TYPE Response_Values :
STRUCT
	Header				:UINT;			// Fixed 0x1234
	Status				:UINT;			// Status word of the sensor and Compute Box
	Fx					:INT;			// X-axis force in 32 bit Counts*
	Fy					:INT;			// Y-axis force in 32 bit Counts*
	Fz					:INT;			// Z-axis force in 32 bit Counts*
	Tx					:INT;			// X-axis torque in 32 bit Counts* (0 if not available)
	Ty					:INT;			// Y-axis torque in 32 bit Counts* (0 if not available)
	Tz					:INT;			// Z-axis torque in 32 bit Counts* (0 if not available)
END_STRUCT
END_TYPE

(* stored: Version 1.1.0.1
   DUT Response_Values: Id {12e477d7-975a-43ec-be38-95f5335893b7} *)
